// TIA Portal V20 export
FUNCTION "V102" : Void   // FC15, FBD
{ S7_Optimized_Access := 'TRUE' }
// stored: SetENOAutomatically false
   VAR_TEMP
      Temp : "DigVal";
      Temp_1 : "DigVal";
      State : "Service_States";
   END_VAR
BEGIN

REGION Network 1: Channel input
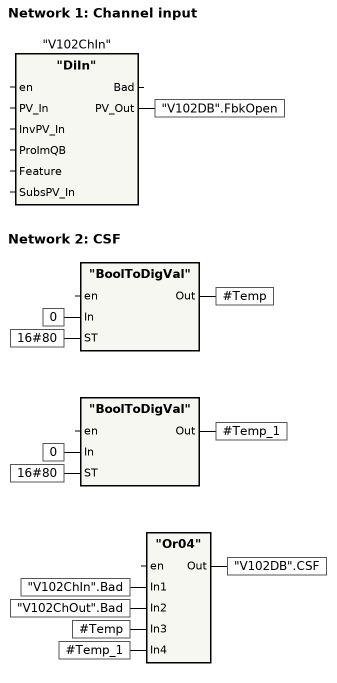
   "V102ChIn"(PV_Out => "V102DB".FbkOpen);   // "DiIn"
END_REGION

REGION Network 2: CSF
   "BoolToDigVal"(In := 0, ST := 16#80, Out => #Temp);
   "BoolToDigVal"(In := 0, ST := 16#80, Out => #Temp_1);
   "Or04"(In1 := "V102ChIn".Bad, In2 := "V102ChOut".Bad, In3 := #Temp, In4 := #Temp_1, Out => "V102DB".CSF);
END_REGION

REGION Network 3: VlvAn Intlock
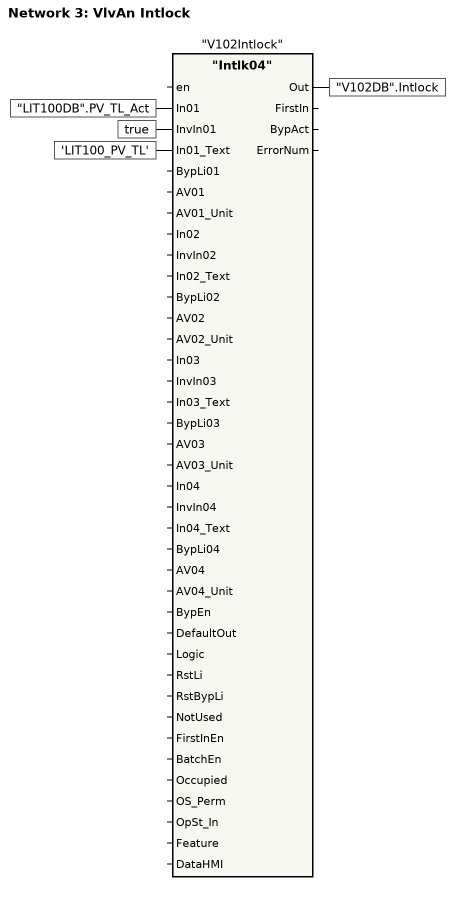
   "V102Intlock"(In01 := "LIT100DB".PV_TL_Act,   // "Intlk04"
                 InvIn01 := true,
                 In01_Text := 'LIT100_PV_TL',
                 Out => "V102DB".Intlock);
END_REGION

REGION Network 4: VlvAnL
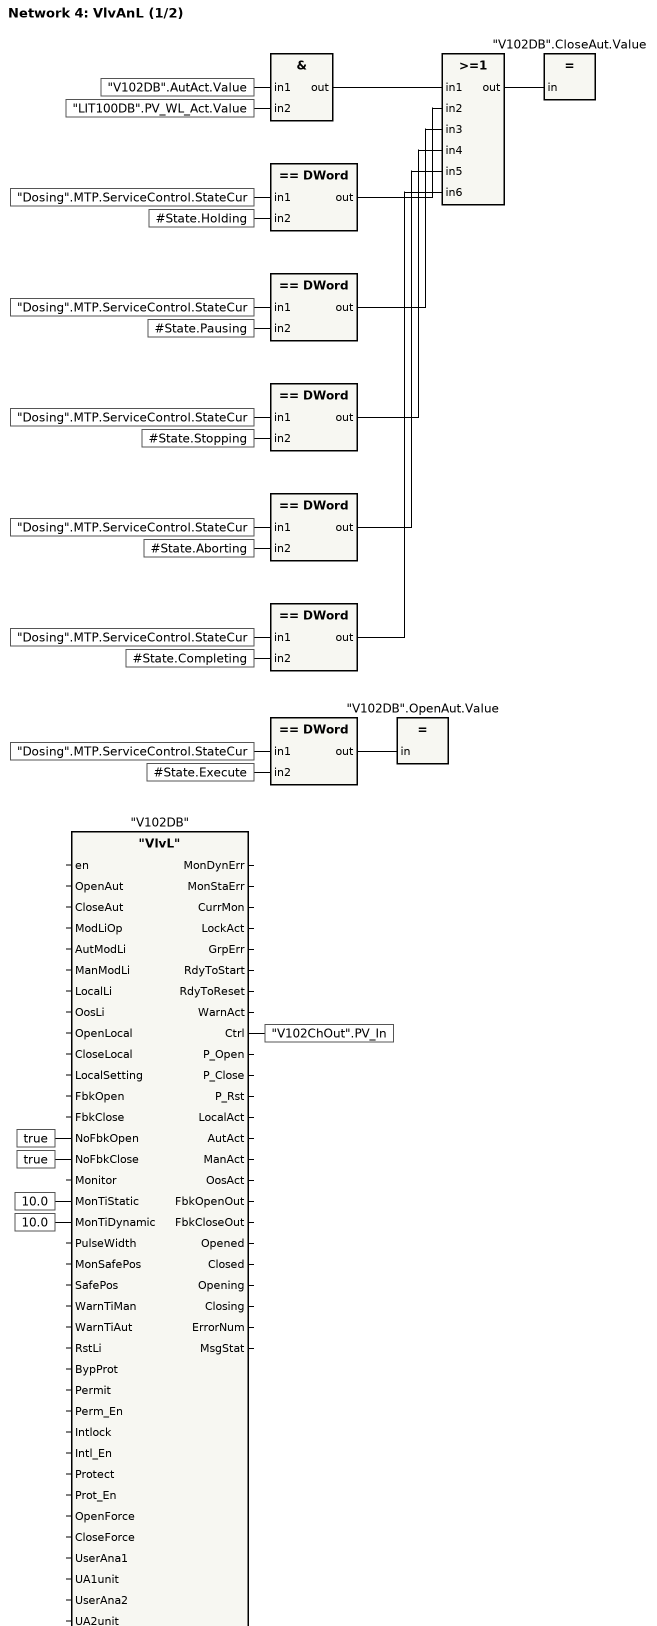
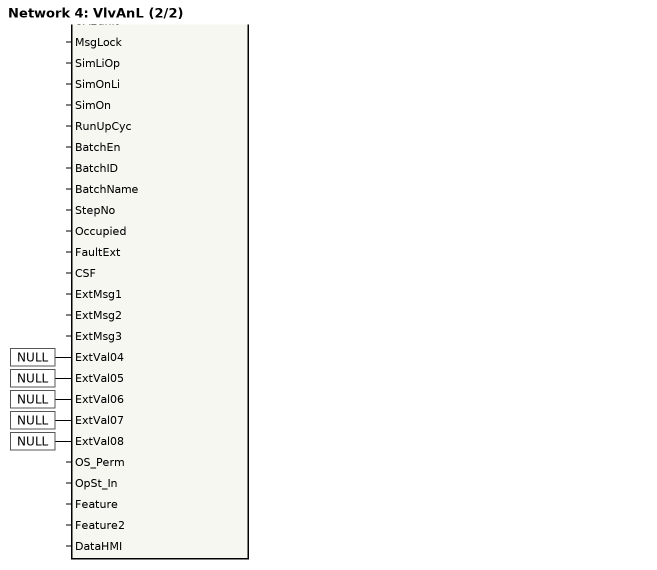
   "V102DB".CloseAut.Value := ("V102DB".AutAct.Value AND "LIT100DB".PV_WL_Act.Value) OR ("Dosing".MTP.ServiceControl.StateCur = #State.Holding) OR ("Dosing".MTP.ServiceControl.StateCur = #State.Pausing) OR ("Dosing".MTP.ServiceControl.StateCur = #State.Stopping) OR ("Dosing".MTP.ServiceControl.StateCur = #State.Aborting) OR ("Dosing".MTP.ServiceControl.StateCur = #State.Completing);
   "V102DB".OpenAut.Value := "Dosing".MTP.ServiceControl.StateCur = #State.Execute;
   "V102DB"(NoFbkOpen := true,   // "VlvL"
            NoFbkClose := true,
            MonTiStatic := 10.0,
            MonTiDynamic := 10.0,
            ExtVal04 := NULL,
            ExtVal05 := NULL,
            ExtVal06 := NULL,
            ExtVal07 := NULL,
            ExtVal08 := NULL,
            Ctrl => "V102ChOut".PV_In);
END_REGION

REGION Network 5: MTP
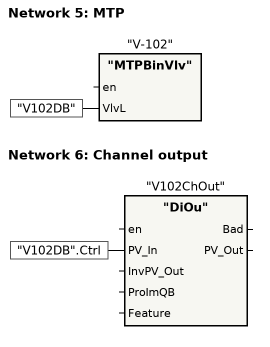
   "V-102"(VlvL := "V102DB");   // "MTPBinVlv"
END_REGION

REGION Network 6: Channel output
   "V102ChOut"(PV_In := "V102DB".Ctrl);   // "DiOu"
END_REGION
END_FUNCTION
